{attribute 'qualified_only'}
TYPE E_Module_Fault :
(
    None := 0,
    GenericFault,
    NotReady,
    Timeout
);
END_TYPE

(* stored: Version 1.1.0.1, ProductVersion 3.1.4024.13
   DUT E_Module_Fault: Id {ee34969d-7d09-4397-a8e0-02a1b77554fb} *)
